{attribute 'reflection'}
FUNCTION_BLOCK PUBLIC ABSTRACT FB_FunctionBase EXTENDS FB_Base
VAR_OUTPUT
	sActiveState	: STRING 		:= 'Idle'	; // active state of device 
	bManual			: BOOL 			:= FALSE 	; // device is in manual mode
	bIsSafe			: BOOL 			:= FALSE	; // Device is locked and safe
	bHeld			: BOOL 			:= FALSE 	; // Function is held
	bBlockedCommand	: BOOL 			:= FALSE 	; // a device command is blocked because of collision detect 
END_VAR
VAR
	bCmdManual 		: BOOL			:= FALSE	; // manual commands enabled control functions (thus disable automatic)
END_VAR

SUPER^();

// Communicate active state
IF bErrorActive THEN 
	sActiveState := TO_STRING(stFault.Description);
ELSIF NOT bInitOk THEN 
	sActiveState := 'Not initialized';
ELSIF bManual THEN 
	sActiveState := 'Manual operation';
ELSE
	sActiveState := 'Operational';
END_IF 

// Set manual command mode
bManual := bCmdManual;

// Execute device functions
IF bInitOk THEN  
	ExecMachineSafety();
	ExecDevFunctions();
END_IF

// Set fault if commands are blocked
IF bBlockedCommand AND bHeld THEN 
	stFault.Active 			:= TRUE ;
	stFault.Description		:= 'Function is blocked';
	stFault.FaultType		:= E_FaultTypes.MC;
END_IF

METHOD PUBLIC CmdHold : BOOL
VAR_INPUT
END_VAR
bHeld 	:= TRUE ;
CmdHold := bHeld ;
END_METHOD

METHOD PUBLIC CmdManual : BOOL
VAR_INPUT
END_VAR
// Enable manual mode
bCmdManual := TRUE;
END_METHOD

METHOD PUBLIC CmdSafeStop : BOOL
VAR_INPUT
END_VAR
// check if device is safe
bIsSafe 	:= NOT bEnable ;
CmdSafeStop := bIsSafe ;
END_METHOD

METHOD PROTECTED ExecDevFunctions : BOOL
VAR_INPUT
END_VAR
END_METHOD

METHOD PROTECTED ExecMachineSafety : BOOL
VAR_INPUT
END_VAR
END_METHOD

END_FUNCTION_BLOCK

(* stored: Version 1.1.0.1, ProductVersion 3.1.4024.11
   POU FB_FunctionBase: Id {ef86906a-1986-411c-841b-bedecc286c14}, SpecialFunc None
   Method CmdHold: Id {b7b43511-9b6a-4b39-b79c-935cd576f467}
   Method CmdManual: Id {a80209b9-b449-43b8-997f-3d83541a6746}
   Method CmdSafeStop: Id {507980d7-bd9e-492d-a4cc-cc2ab03b31c7}
   Method ExecDevFunctions: Id {351765c3-accd-4b4a-927f-08fd149221ad}
   Method ExecMachineSafety: Id {21d44c79-19d0-4d2a-975d-6d59086163c6} *)
